
FUNCTION CB_byte_to_word : WORD

TITLE = ' Convert a byte into a word '
VERSION : '1.0'
AUTHOR  : CB
NAME    : bytToWor
FAMILY  : TNI

VAR_INPUT
    IN : BYTE;
END_VAR

BEGIN

CB_byte_to_word := IN;

END_FUNCTION
